Staubli VAL3: delete.pgx

public program delete(num x_nIndexGun)
begin
  $ddel(saveTool:gun,x_nIndexGun)
  $ddel(saveTool:name,x_nIndexGun)
  $ddel(saveTool:sActionOFF,x_nIndexGun)
  $ddel(saveTool:sActionON,x_nIndexGun)
end
